// Mitsubishi GX Works2 project: Dao_Chieu_Chay_Theo_Thoi_Gian   PLC: FX2N/FX2NC

PROGRAM MAIN
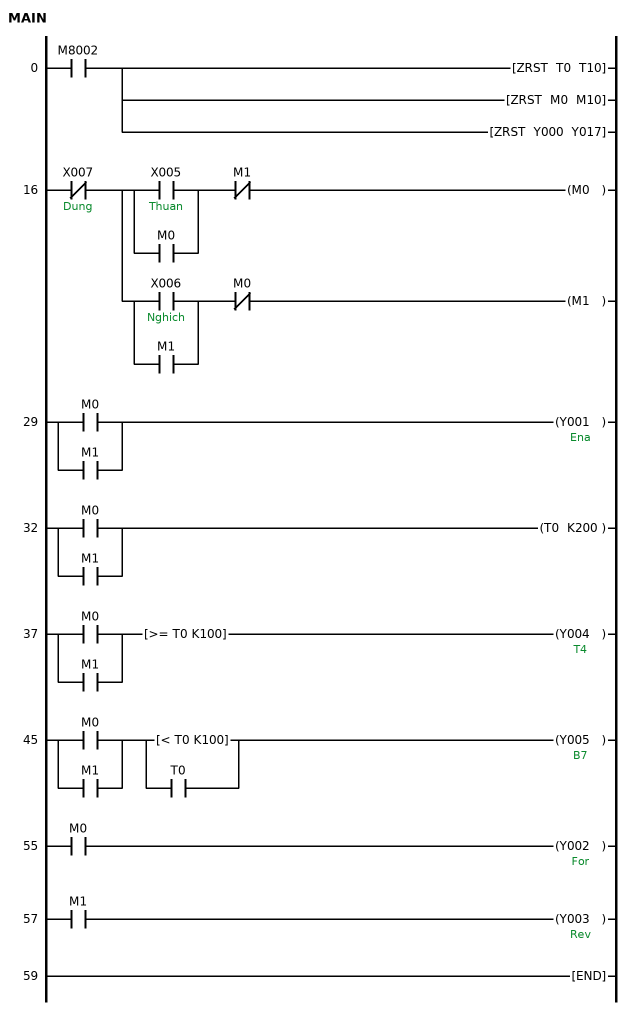
0     LD      M8002
      ZRST    T0 T10
      ZRST    M0 M10
      ZRST    Y000 Y017
16    LDI     X007  ; Dung
      MPS
      LD      X005  ; Thuan
      OR      M0
      ANB
      ANI     M1
      OUT     M0
      MPP
      LD      X006  ; Nghich
      OR      M1
      ANB
      ANI     M0
      OUT     M1
29    LD      M0
      OR      M1
      OUT     Y001  ; Ena
32    LD      M0
      OR      M1
      OUT     T0 K200
37    LD      M0
      OR      M1
      AND>=   T0 K100
      OUT     Y004  ; T4
45    LD      M0
      OR      M1
      LD<     T0 K100
      OR      T0
      ANB
      OUT     Y005  ; B7
55    LD      M0
      OUT     Y002  ; For
57    LD      M1
      OUT     Y003  ; Rev
59    END
END_PROGRAM
